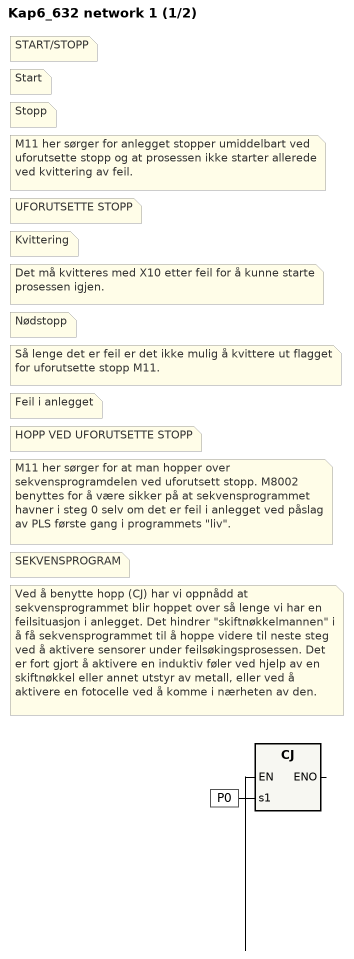
(* [picture p24: structured ladder/FBD of Kap6_632, networks 1 to 1] *)
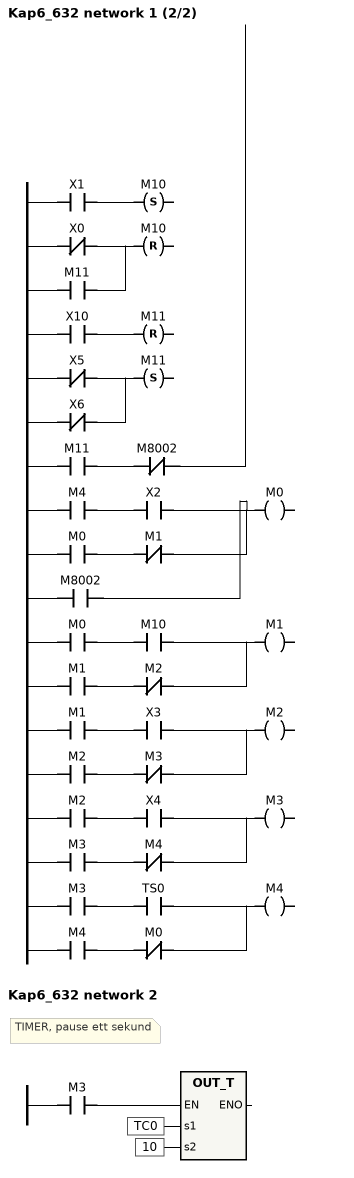
(* network 1 *)
(* START/STOPP *)
(* Start *)
(* Stopp *)
(* M11 her sørger for anlegget stopper umiddelbart ved uforutsette stopp og at prosessen ikke starter allerede ved kvittering av feil. *)
(* UFORUTSETTE STOPP *)
(* Kvittering *)
(* Det må kvitteres med X10 etter feil for å kunne starte prosessen igjen. *)
(* Nødstopp *)
(* Så lenge det er feil er det ikke mulig å kvittere ut flagget for uforutsette stopp M11. *)
(* Feil i anlegget *)
(* HOPP VED UFORUTSETTE STOPP *)
(* M11 her sørger for at man hopper over sekvensprogramdelen ved uforutsett stopp. M8002 benyttes for å være sikker på at sekvensprogrammet havner i steg 0 selv om det er feil i anlegget ved påslag av PLS første gang i programmets "liv". *)
(* SEKVENSPROGRAM *)
(* Ved å benytte hopp (CJ) har vi oppnådd at sekvensprogrammet blir hoppet over så lenge vi har en feilsituasjon i anlegget. Det hindrer "skiftnøkkelmannen" i å få sekvensprogrammet til å hoppe videre til neste steg ved å aktivere sensorer under feilsøkingsprosessen. Det er fort gjort å aktivere en induktiv føler ved hjelp av en skiftnøkkel eller annet utstyr av metall, eller ved å aktivere en fotocelle ved å komme i nærheten av den. *)
SET(X1, M10);
RST((NOT X0) OR M11, M10);
RST(X10, M11);
SET((NOT X5) OR (NOT X6), M11);
CJ(M11 AND NOT M8002, P0);
M0 := (M4 AND X2) OR (M0 AND NOT M1) OR M8002;
M1 := (M0 AND M10) OR (M1 AND NOT M2);
M2 := (M1 AND X3) OR (M2 AND NOT M3);
M3 := (M2 AND X4) OR (M3 AND NOT M4);
M4 := (M3 AND TS0) OR (M4 AND NOT M0);
(* network 2 P0: *)
(* TIMER, pause ett sekund *)
OUT_T(M3, TC0, 10);
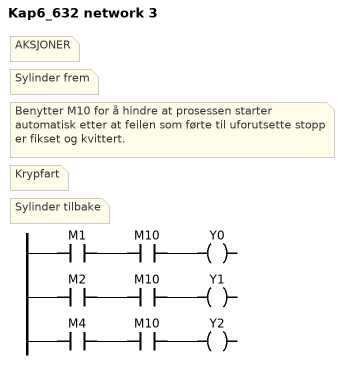
(* network 3 *)
(* AKSJONER *)
(* Sylinder frem *)
(* Benytter M10 for å hindre at prosessen starter automatisk etter at feilen som førte til uforutsette stopp er fikset og kvittert. *)
(* Krypfart *)
(* Sylinder tilbake *)
Y0 := M1 AND M10;
Y1 := M2 AND M10;
Y2 := M4 AND M10;
END_PROGRAM

PROGRAM Kap6_633
(* structured ladder/FBD written out as ST: instructions are called as NAME(EN, inputs, outputs); _pN, _eN, _tN stand for wires *)
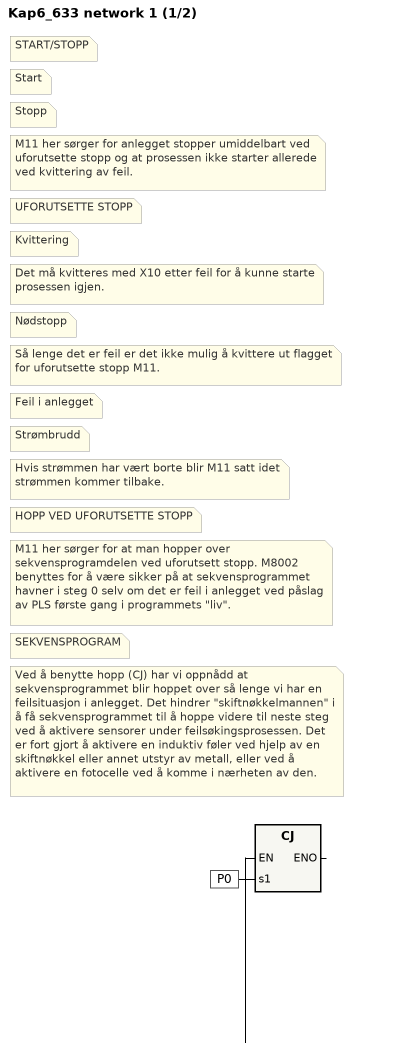
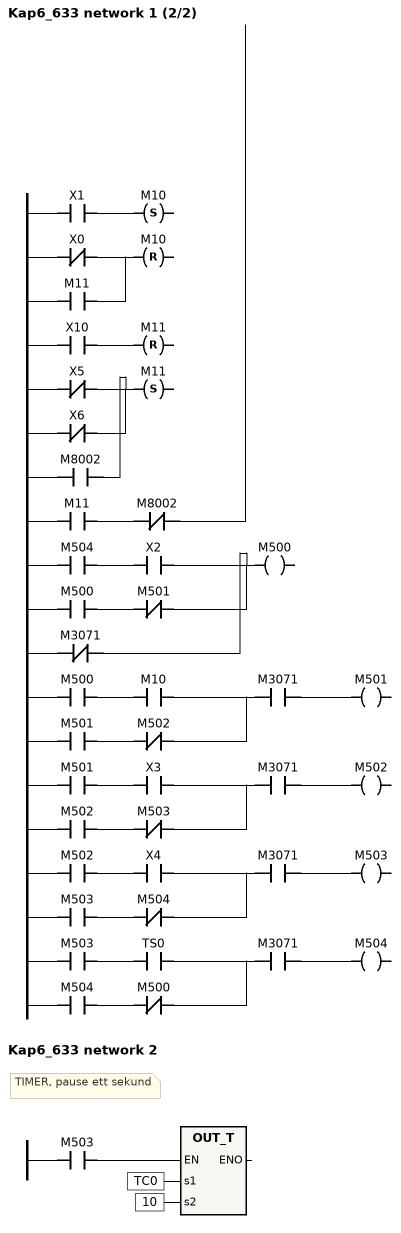
(* network 1 *)
(* START/STOPP *)
(* Start *)
(* Stopp *)
(* M11 her sørger for anlegget stopper umiddelbart ved uforutsette stopp og at prosessen ikke starter allerede ved kvittering av feil. *)
(* UFORUTSETTE STOPP *)
(* Kvittering *)
(* Det må kvitteres med X10 etter feil for å kunne starte prosessen igjen. *)
(* Nødstopp *)
(* Så lenge det er feil er det ikke mulig å kvittere ut flagget for uforutsette stopp M11. *)
(* Feil i anlegget *)
(* Strømbrudd *)
(* Hvis strømmen har vært borte blir M11 satt idet strømmen kommer tilbake. *)
(* HOPP VED UFORUTSETTE STOPP *)
(* M11 her sørger for at man hopper over sekvensprogramdelen ved uforutsett stopp. M8002 benyttes for å være sikker på at sekvensprogrammet havner i steg 0 selv om det er feil i anlegget ved påslag av PLS første gang i programmets "liv". *)
(* SEKVENSPROGRAM *)
(* Ved å benytte hopp (CJ) har vi oppnådd at sekvensprogrammet blir hoppet over så lenge vi har en feilsituasjon i anlegget. Det hindrer "skiftnøkkelmannen" i å få sekvensprogrammet til å hoppe videre til neste steg ved å aktivere sensorer under feilsøkingsprosessen. Det er fort gjort å aktivere en induktiv føler ved hjelp av en skiftnøkkel eller annet utstyr av metall, eller ved å aktivere en fotocelle ved å komme i nærheten av den. *)
SET(X1, M10);
RST((NOT X0) OR M11, M10);
RST(X10, M11);
SET((NOT X5) OR (NOT X6) OR M8002, M11);
CJ(M11 AND NOT M8002, P0);
M500 := (M504 AND X2) OR (M500 AND NOT M501) OR (NOT M3071);
M501 := ((M500 AND M10) OR (M501 AND NOT M502)) AND M3071;
M502 := ((M501 AND X3) OR (M502 AND NOT M503)) AND M3071;
M503 := ((M502 AND X4) OR (M503 AND NOT M504)) AND M3071;
M504 := ((M503 AND TS0) OR (M504 AND NOT M500)) AND M3071;
(* network 2 P0: *)
(* TIMER, pause ett sekund *)
OUT_T(M503, TC0, 10);
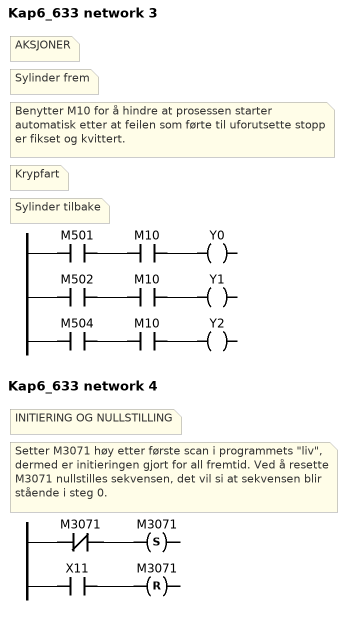
(* network 3 *)
(* AKSJONER *)
(* Sylinder frem *)
(* Benytter M10 for å hindre at prosessen starter automatisk etter at feilen som førte til uforutsette stopp er fikset og kvittert. *)
(* Krypfart *)
(* Sylinder tilbake *)
Y0 := M501 AND M10;
Y1 := M502 AND M10;
Y2 := M504 AND M10;
(* network 4 *)
(* INITIERING OG NULLSTILLING *)
(* Setter M3071 høy etter første scan i programmets "liv", dermed er initieringen gjort for all fremtid. Ved å resette M3071 nullstilles sekvensen, det vil si at sekvensen blir stående i steg 0. *)
SET(NOT M3071, M3071);
RST(X11, M3071);
END_PROGRAM

PROGRAM Kap6_652
(* structured ladder/FBD written out as ST: instructions are called as NAME(EN, inputs, outputs); _pN, _eN, _tN stand for wires *)
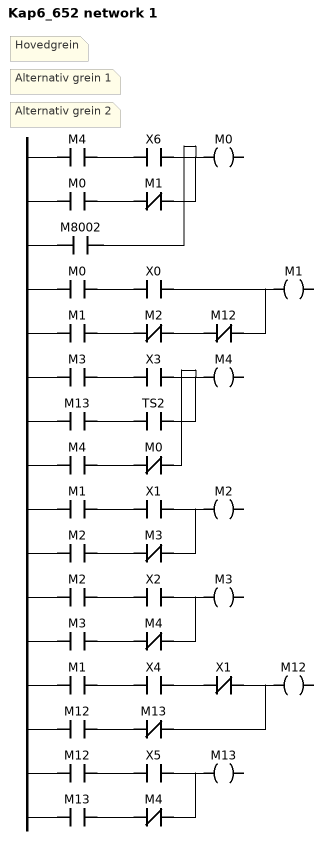
(* network 1 *)
(* Hovedgrein *)
(* Alternativ grein 1 *)
(* Alternativ grein 2 *)
M0 := (M4 AND X6) OR (M0 AND NOT M1) OR M8002;
M1 := (M0 AND X0) OR (M1 AND NOT M2 AND NOT M12);
M4 := (M3 AND X3) OR (M13 AND TS2) OR (M4 AND NOT M0);
M2 := (M1 AND X1) OR (M2 AND NOT M3);
M3 := (M2 AND X2) OR (M3 AND NOT M4);
M12 := (M1 AND X4 AND NOT X1) OR (M12 AND NOT M13);
M13 := (M12 AND X5) OR (M13 AND NOT M4);
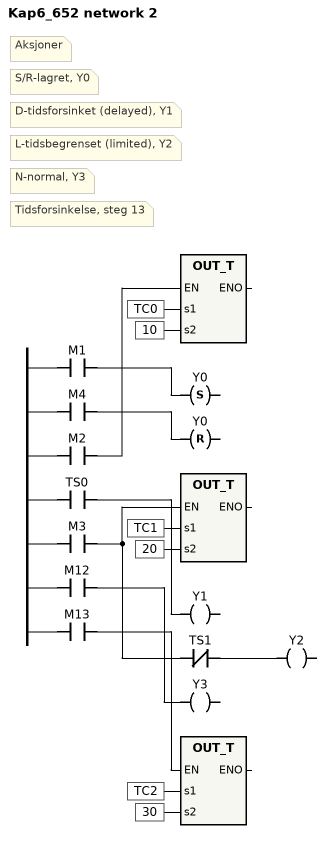
(* network 2 *)
(* Aksjoner *)
(* S/R-lagret, Y0 *)
(* D-tidsforsinket (delayed), Y1 *)
(* L-tidsbegrenset (limited), Y2 *)
(* N-normal, Y3 *)
(* Tidsforsinkelse, steg 13 *)
SET(M1, Y0);
RST(M4, Y0);
OUT_T(M2, TC0, 10);
Y1 := TS0;
Y2 := M3 AND NOT TS1;
OUT_T(M3, TC1, 20);
Y3 := M12;
OUT_T(M13, TC2, 30);
END_PROGRAM

PROGRAM Kap6_654
(* structured ladder/FBD written out as ST: instructions are called as NAME(EN, inputs, outputs); _pN, _eN, _tN stand for wires *)
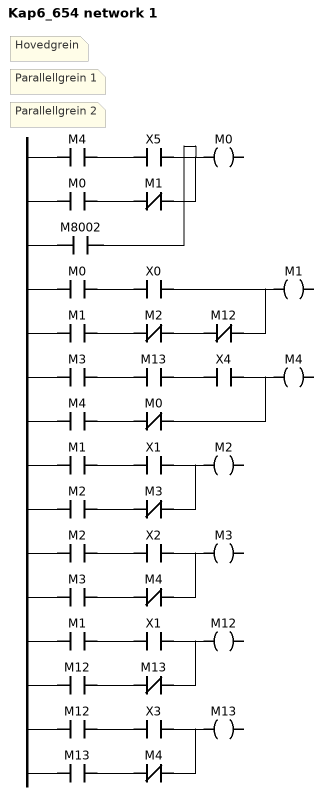
(* network 1 *)
(* Hovedgrein *)
(* Parallellgrein 1 *)
(* Parallellgrein 2 *)
M0 := (M4 AND X5) OR (M0 AND NOT M1) OR M8002;
M1 := (M0 AND X0) OR (M1 AND NOT M2 AND NOT M12);
M4 := (M3 AND M13 AND X4) OR (M4 AND NOT M0);
M2 := (M1 AND X1) OR (M2 AND NOT M3);
M3 := (M2 AND X2) OR (M3 AND NOT M4);
M12 := (M1 AND X1) OR (M12 AND NOT M13);
M13 := (M12 AND X3) OR (M13 AND NOT M4);
END_PROGRAM

PROGRAM Kap6_656
(* structured ladder/FBD written out as ST: instructions are called as NAME(EN, inputs, outputs); _pN, _eN, _tN stand for wires *)
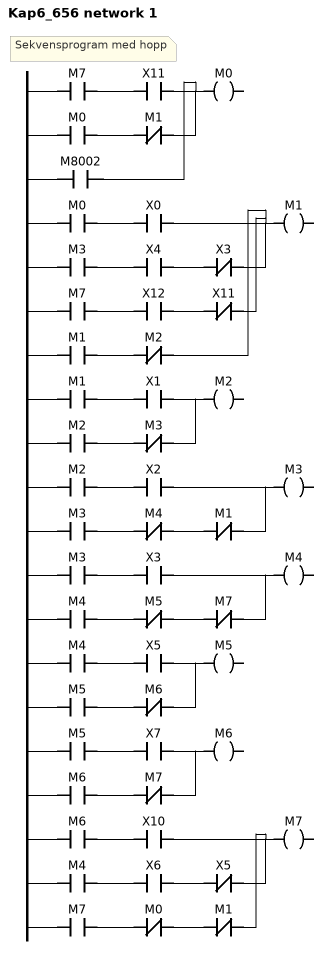
(* network 1 *)
(* Sekvensprogram med hopp *)
M0 := (M7 AND X11) OR (M0 AND NOT M1) OR M8002;
M1 := (M0 AND X0) OR (M3 AND X4 AND NOT X3) OR (M7 AND X12 AND NOT X11) OR (M1 AND NOT M2);
M2 := (M1 AND X1) OR (M2 AND NOT M3);
M3 := (M2 AND X2) OR (M3 AND NOT M4 AND NOT M1);
M4 := (M3 AND X3) OR (M4 AND NOT M5 AND NOT M7);
M5 := (M4 AND X5) OR (M5 AND NOT M6);
M6 := (M5 AND X7) OR (M6 AND NOT M7);
M7 := (M6 AND X10) OR (M4 AND X6 AND NOT X5) OR (M7 AND NOT M0 AND NOT M1);
END_PROGRAM

PROGRAM Kap5_5422
(* structured ladder/FBD written out as ST: instructions are called as NAME(EN, inputs, outputs); _pN, _eN, _tN stand for wires *)
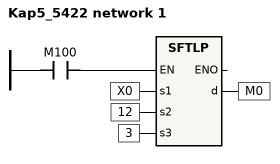
(* network 1 *)
SFTLP(M100, X0, 12, 3, M0);
END_PROGRAM

PROGRAM Kap3_332
(* structured ladder/FBD written out as ST: instructions are called as NAME(EN, inputs, outputs); _pN, _eN, _tN stand for wires *)
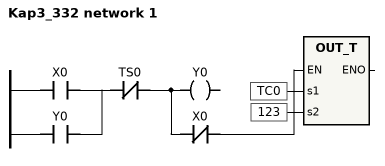
(* network 1 *)
_p1 := (X0 OR Y0) AND NOT TS0;
Y0 := _p1;
OUT_T(_p1 AND NOT X0, TC0, 123);
END_PROGRAM

PROGRAM Kap4_422
(* structured ladder/FBD written out as ST: instructions are called as NAME(EN, inputs, outputs); _pN, _eN, _tN stand for wires *)
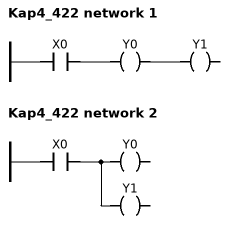
(* network 1 *)
Y0 := X0;
Y1 := X0;
(* network 2 *)
Y0 := X0;
Y1 := X0;
END_PROGRAM

PROGRAM Kap4_441
(* structured ladder/FBD written out as ST: instructions are called as NAME(EN, inputs, outputs); _pN, _eN, _tN stand for wires *)
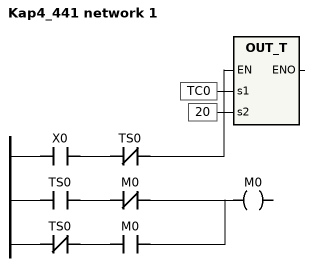
(* network 1 *)
OUT_T(X0 AND NOT TS0, TC0, 20);
M0 := (TS0 AND NOT M0) OR (NOT TS0 AND M0);
END_PROGRAM

PROGRAM Kap4_461
(* structured ladder/FBD written out as ST: instructions are called as NAME(EN, inputs, outputs); _pN, _eN, _tN stand for wires *)
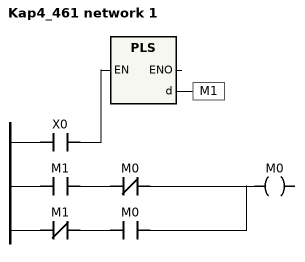
(* network 1 *)
PLS(X0, M1);
M0 := (M1 AND NOT M0) OR (NOT M1 AND M0);
END_PROGRAM

PROGRAM Kap5_531
VAR
  Data10 : DINT;
  Data12 : DINT;
END_VAR
(* structured ladder/FBD written out as ST: instructions are called as NAME(EN, inputs, outputs); _pN, _eN, _tN stand for wires *)
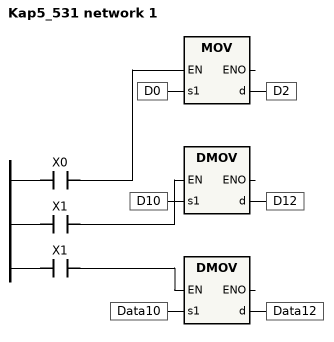
(* network 1 *)
MOV(X0, D0, D2);
DMOV(X1, D10, D12);
DMOV(X1, Data10, Data12);
END_PROGRAM

PROGRAM Kap5_532
(* structured ladder/FBD written out as ST: instructions are called as NAME(EN, inputs, outputs); _pN, _eN, _tN stand for wires *)
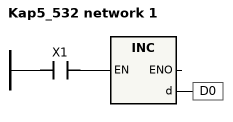
(* network 1 *)
INC(X1, D0);
END_PROGRAM

PROGRAM Kap5_533
(* structured ladder/FBD written out as ST: instructions are called as NAME(EN, inputs, outputs); _pN, _eN, _tN stand for wires *)
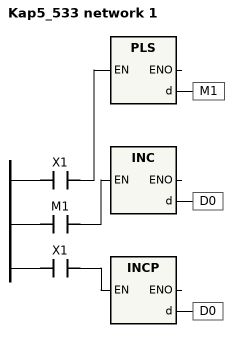
(* network 1 *)
PLS(X1, M1);
INC(M1, D0);
INCP(X1, D0);
END_PROGRAM

PROGRAM Kap5_534
(* structured ladder/FBD written out as ST: instructions are called as NAME(EN, inputs, outputs); _pN, _eN, _tN stand for wires *)
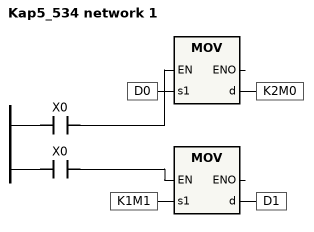
(* network 1 *)
MOV(X0, D0, K2M0);
MOV(X0, K1M1, D1);
END_PROGRAM

PROGRAM Kap5_541
VAR
  Data1 : INT;
  Data2 : INT;
  Data3 : INT;
END_VAR
(* structured ladder/FBD written out as ST: instructions are called as NAME(EN, inputs, outputs); _pN, _eN, _tN stand for wires *)
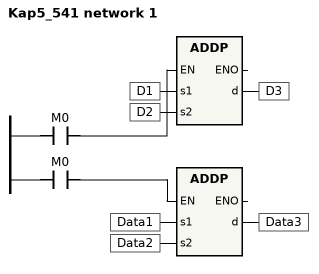
(* network 1 *)
ADDP(M0, D1, D2, D3);
ADDP(M0, Data1, Data2, Data3);
END_PROGRAM

PROGRAM Kap5_542
VAR
  Data4 : DINT;
  Data6 : DINT;
  Data8 : DINT;
END_VAR
(* structured ladder/FBD written out as ST: instructions are called as NAME(EN, inputs, outputs); _pN, _eN, _tN stand for wires *)
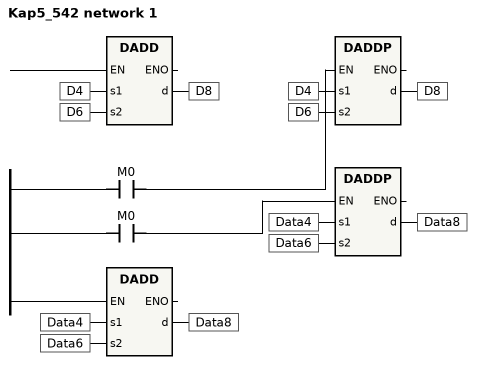
(* network 1 *)
DADD(TRUE, D4, D6, D8);
DADD(TRUE, Data4, Data6, Data8);
DADDP(M0, D4, D6, D8);
DADDP(M0, Data4, Data6, Data8);
END_PROGRAM

PROGRAM Kap5_543
VAR
  Data1 : INT;
  Data2 : INT;
  Data3 : INT;
END_VAR
(* structured ladder/FBD written out as ST: instructions are called as NAME(EN, inputs, outputs); _pN, _eN, _tN stand for wires *)
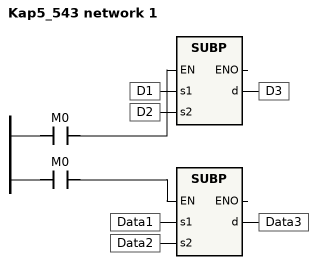
(* network 1 *)
SUBP(M0, D1, D2, D3);
SUBP(M0, Data1, Data2, Data3);
END_PROGRAM

PROGRAM Kap5_544
VAR
  Data4 : DINT;
  Data6 : DINT;
  Data8 : DINT;
END_VAR
(* structured ladder/FBD written out as ST: instructions are called as NAME(EN, inputs, outputs); _pN, _eN, _tN stand for wires *)
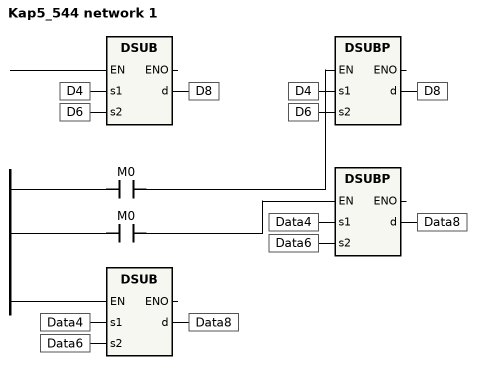
(* network 1 *)
DSUB(TRUE, D4, D6, D8);
DSUB(TRUE, Data4, Data6, Data8);
DSUBP(M0, D4, D6, D8);
DSUBP(M0, Data4, Data6, Data8);
END_PROGRAM

PROGRAM Kap5_545
VAR
  Data1 : INT;
  Data2 : INT;
  Data3 : DINT;
END_VAR
(* structured ladder/FBD written out as ST: instructions are called as NAME(EN, inputs, outputs); _pN, _eN, _tN stand for wires *)
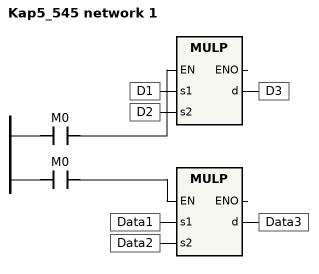
(* network 1 *)
MULP(M0, D1, D2, D3);
MULP(M0, Data1, Data2, Data3);
END_PROGRAM

PROGRAM Kap5_546
VAR
  Data4 : DINT;
  Data6 : DINT;
  Data8 : ARRAY [0..1] OF DINT;
END_VAR
(* structured ladder/FBD written out as ST: instructions are called as NAME(EN, inputs, outputs); _pN, _eN, _tN stand for wires *)
